{attribute 'linkalways'} 
{attribute 'no_explicit_call' := 'This FB is a CLASS and must be accessed using methods or properties'}
{attribute 'enable_dynamic_creation'}
FUNCTION_BLOCK FINAL MIN_REAL EXTENDS Node
VAR
	in1 : _REAL(0.0);
	in2 : _REAL(0.0);
	out : _REAL(0.0);
END_VAR

METHOD PUBLIC Clone : I_Node
VAR
	pNode : POINTER TO MIN_REAL;
END_VAR
pNode := __NEW(MIN_REAL);
Clone := pNode^;
END_METHOD

METHOD FB_init : BOOL
VAR_INPUT
	bInitRetains : BOOL; // if TRUE, the retain variables are initialized (warm start / cold start)
	bInCopyCode : BOOL;  // if TRUE, the instance afterwards gets moved into the copy code (online change)
END_VAR
AddInput('in1',THIS^.in1);
AddInput('in2',THIS^.in2);
AddOutput('out', THIS^.out);
END_METHOD

METHOD PROTECTED OnExecute
VAR
END_VAR
out.Value := MIN(in1.Value, in2.Value);
END_METHOD

END_FUNCTION_BLOCK

(* stored: Version 1.1.0.1, ProductVersion 3.1.4024.15
   POU MIN_REAL: Id {7f5e24fa-a12e-4221-bd25-bcfca6eb7ed0}, SpecialFunc None
   Folder Constructor: Id {c05c00c4-7195-4fc7-aeb7-2d56ca0b1f41}
   Method Clone: Id {3da4f1ce-1f2c-4e4d-a7ae-0a85321a5ea9}
   Method FB_init: Id {7307681f-7f2f-4e77-add0-de352ea3ae0e}
   Method OnExecute: Id {989a5c16-259b-4df9-b7a8-6cab81d0770d} *)
